FUNCTION_BLOCK Test_WriteBySymbolName_KeepingHandle EXTENDS T_UnitTestBase
VAR
    AdsWriteBySymbolName : T_AdsWriteBySymbolName;
    ValueToWrite : INT := 3456;
    WriteResult : INT;
    ScanCount : DINT;
END_VAR

CASE State OF
    0:
        ValueToWrite := 3456;
        WriteResult := 0;
        ScanCount := 0;
    
        AdsWriteBySymbolName.Execute(
            AmsNetId:= '', 
            Port:= Constants.PortNo, 
            SymbolName:= 'PB_TestRunner.Test_WriteBySymbolName_KeepingHandle.WriteResult', 
            WriteDataAddress:= ADR(ValueToWrite), 
            WriteDataLength:= SIZEOF(ValueToWrite), 
            KeepSymbolHandle:= TRUE);

        State := 10;
        
    10:
        ScanCount := ScanCount + 1;
        IF NOT AdsWriteBySymbolName.Execution.Busy THEN
            State := 20;    
		END_IF
        
    20:
        Assertion.AssertEquals_INT(
            Expected     := 3456,
            Actual       := WriteResult,
            Variablename := 'WriteResult'); 
 
        TestFinished();
        State := 0;
END_CASE

AdsWriteBySymbolName();

END_FUNCTION_BLOCK

(* stored: Version 1.1.0.1, ProductVersion 3.1.4024.9
   POU Test_WriteBySymbolName_KeepingHandle: Id {0212d425-6247-0e8e-2cf6-15279713d8f0}, SpecialFunc None *)
